// TIA Portal V17 program export: 0 tag tables, 0 data types, 0 data blocks, 2 code blocks (in call order from the OBs), 0 instance data blocks

ORGANIZATION_BLOCK "Main"   // OB1, LAD, ProgramCycle
TITLE = "Main Program Sweep (Cycle)"
{ S7_Optimized_Access := 'TRUE' }
VERSION : 0.1
// stored: AutoNumber true, IsIECCheckEnabled false, SetENOAutomatically false
   VAR_INPUT
      Initial_Call : Bool;   // Initial call of this OB
      Remanence : Bool;   // =True, if remanent data are available
   END_VAR
BEGIN

REGION Network 1
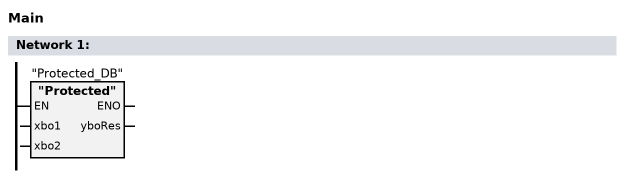
   RUNG wire#powerrail
      "Protected_DB"(xbo1 :=, xbo2 :=, yboRes =>)
   END_RUNG
   // the same network as SCL:
   "Protected_DB"();   // "Protected"
END_REGION
END_ORGANIZATION_BLOCK

FUNCTION "Add" : Void
{ S7_Optimized_Access := 'TRUE' }
VERSION : 0.1
   VAR_INPUT 
      xreVal1 : Real;
      xreVal : Real;
   END_VAR

   VAR_OUTPUT 
      yreResult : Real;
   END_VAR


BEGIN
	#yreResult := #xreVal1 + #xreVal2;
END_FUNCTION
